// TIA Portal project "HMI_design" (V15)

(* hardware
DEVICE "PC-System_1"  SIMATIC PC station
   slot 0: "SIMATIC PC station"  Rail  SIMATIC PC-Station  V1.0
      slot 125: "Stationmanager"  Station_Manager  V6.0.4
   slot 1: "HMI_RT_1"  WinCC RT Advanced  6AV2 104-0xxxx-xxxx  15.0.0.0
      slot 33792: "Host interface"  Host interface
   slot 2: "IE general_1"  IE General  IE_CP  V8.2.0
DEVICE "S7-1200 station_1"  S7-1200 Station
   slot 0: "Rack_0"  S7-1200 Rack  Rack  V1.0
   slot 1: "PLC_1"  CPU 1214C DC/DC/DC  6ES7 214-1AG40-0XB0  V4.2
*)

// ===== PLC "PLC_1"  CPU 1214C DC/DC/DC =====

VAR_GLOBAL   // PLC tag table "Default tag table"
   "ON" AT %I0.0 : Bool;
   "OFF" AT %I0.1 : Bool;
   "LIGHT" AT %Q0.0 : Bool;
   "Value" AT %MW10 : UInt;
END_VAR

ORGANIZATION_BLOCK "Main"   // OB1, LAD, ProgramCycle
TITLE = "Main Program Sweep (Cycle)"
{ S7_Optimized_Access := 'TRUE' }
VERSION : 0.1
   VAR_INPUT
      Initial_Call : Bool;   // Initial call of this OB
      Remanence : Bool;   // =True, if remanent data are available
   END_VAR
BEGIN

REGION Network 1
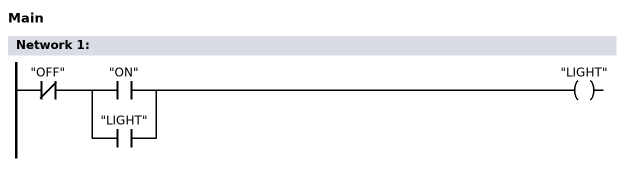
   RUNG wire#powerrail
      I_Contact( "OFF" )
      wire#w1
      Contact( "ON" )
      wire#w2
      Coil( "LIGHT" )
   END_RUNG
   RUNG wire#w1
      Contact( "LIGHT" )
   END_RUNG wire#w2
   // the same network as SCL:
   "LIGHT" := NOT "OFF" AND ("ON" OR "LIGHT");
END_REGION
END_ORGANIZATION_BLOCK

(* ===== HMI "HMI_RT_1" =====
system functions are stored by id; their names below are inferred from use
connection "HMI_Connection_1": ETHERNET, S7_1200_OMS

HMI tags "Default tag table"
   "ON" : Bool = PLC ON AT %I0.0, 1 s
   "OFF" : Bool = PLC OFF AT %I0.1, 1 s
   "LIGHT" : Bool = PLC LIGHT AT %Q0.0, 1 s
   "Value" : UInt = PLC Value AT %MW10, 1 s

screen "Manual" 1024x768
   TextField "Text field_1" at 313,10 size 188x62; Text 'Manual'

screen "Set up" 1024x768
   TextField "Text field_1" at 313,10 size 188x62; Text 'Set up'

screen "Start up" 1024x768
   TextField "Text field_1" at 313,10 size 188x62; Text 'Start up'
   Button "Button_1" at 285,131 size 96x32; TextOff 'ON'; Authorization "Operate"
      on Press: SetBit("ON")
      on Release: ResetBit("ON")
   Button "Button_2" at 285,192 size 96x32; TextOff 'OFF'; Authorization "Configure"
      on Release: ResetBit("OFF")
      on Press: SetBit("OFF")
   Circle "Circle_1" at 501,131 size 85x85
      Appearance <- "LIGHT"
   Button "Button_3" at 679,12 size 47x34; TextOff 'X'
      on Click: StopRuntime(0)
   Button "Button_4" at 46,17 size 110x54; TextOff 'Log Off'
      on Click: function_f23ef4c9()
   IOField "I/O field_1" at 248,242 size 255x76; FormatPattern 9999
      ProcessValue <- "Value"

screen "Login_Screen" 1024x768
   TextField "Text field_1" at 292,2 size 226x86; Text 'Login Screen'
   Button "Button_1" at 316,122 size 177x77; TextOff 'Login'
      on Click: function_a2a04561()
   Button "Button_2" at 610,669 size 146x64; TextOff 'Go to Start up'
   Button "Button_3" at 853,669 size 146x64; TextOff 'Go to Set up'
      on Click: function_cf6f4242(N, -1)
*)